	FUNCTION_BLOCK FB 1026
	TITLE =A_3911_MXZ01MA CHAIN CONVEYOR UNDER KILN 2
	//COPYRIGHT:     (C) 2009  BUHLER AG, CH-9240 UZWIL, SWITZERLAND
	//
	//PRODUCT:       WinCoS_BIW01_09
	//
	//TITLE:         CHAIN CONVEYOR UNDER KILN 2
	//
	//--------------------------------------------------------------------------------
	//
	//IDENT:         AUTHOR:             DEPT:                             DATE:
	//
	//P01_FB1026.1.0 K.Renz              CSB41                             08.Jun.2010
	//               1st Release
	//
	//--------------------------------------------------------------------------------
	//
	//PURPOSE:
	//
	//MANUAL :
	//
	//RESTRICTIONS:
	//
	//--------------------------------------------------------------------------------
	AUTHOR  : KR
	FAMILY  : USW
	VERSION : 0.0


	VAR
	         Ma :  UDT 20500  ;  // Machine
	         A_3911_BQS06 : FB84;  // Mon1: DigInpCont
	         Mon2  : FB14 ;   // Mon2: DigInpCont
	         Mon3  : FB14  ;  // spare
	         A_3911_BSA08 : FB14;  // Mon4: DigInpCont
	         Mon5  : FB14 ;   // spare
	         Mon6  : FB14 ;   // spare
	         A_3911_MXZ01 : FB12; // Motor: Motor
	END_VAR

	BEGIN
	NETWORK
	TITLE =Call SSW
	   UC  FB50
	END_FUNCTION_BLOCK
